// TIA Portal V19 export
VAR_GLOBAL   // PLC tag table "D30"
   D30_Ls_Os1 AT %I1086.0 : Bool;   // 105DI2 - 231A1
   D30_Ls_Os2 AT %I1086.4 : Bool;   // 105DI6 - 231A1
END_VAR
